Universal Robots PolyScope program: OnRobot_Pin_Insertion_Example.urp

Program OnRobot_Pin_Insertion_Example (createdIn=3.3.4.310 lastSavedIn=3.7.0.40195 robotSerialNumber=2014359999 directory=/home/ur/ursim-current/programs/TransferVM/Examples/Pendrive installation=default)
Calibrated DH parameters: a=[0.000125, -0.611383, -0.570393, -0.000092, 0.000088, 0]; d=[0.127903, 2.433032, -6.959421, 4.690192, 0.11563, 0.092223]; alpha=[1.570378, -0.01465, -0.007405, 1.570477, -1.570381, 0]; deltaTheta=[-0.000064, -0.058226, 0.116976, -0.058728, 0.000029, -0.000013]
BeforeStart
  URCap F/T Zero (FT-OnRobot, OnRobot A/S)
Robot Program (runOnlyOnce=true)
  URCap F/T Guard (FT-OnRobot, OnRobot A/S) dataModel(OF_PID=0, FX=0.0, FY=0.0, FZ=0.0, TX=0.0, TY=0.0, TZ=0.0, F3D=50.0, T3D=1.0, ABS=true, COORD=0, INDEX=0, STATE=true, ADVANCED=false, NEEDDIGI=false, NAME=50N & 1Nm)
    MoveJ speed 60 deg/s, acceleration 80 deg/s^2 (useActiveTCP=false)
      Waypoint StartWP: TCP in base x=-120.113 y=-431.763 z=146.073 mm, rx=-0.0012 ry=3.1163 rz=0.0389 rad; joints [-91.713, -98.956, -126.223, -46.295, 91.393, -1.776] deg
    URCap F/T Insert Part (FT-OnRobot, OnRobot A/S) dataModel(SPEED=0.05, DEPTH=0.02, FORCE=3, TORQUE=0.2, NAME=20 mm, LEN=0, DEG=0, SILENT=false, ADVANCED=false, ASTART=10, AEND=30, ALIMIT=0.17453292519943295, ASTRENGTH=0.5, pushingForce=5.0, minDistance=0.02, maxDistance=0.042, advanced=true, generateWarning=true, fx=0.0, cfx=true, fy=0.0, cfy=true, fz=0.0, cfz=true, tx=0.0, ctx=true, ty=0.0, cty=true, ctz=true, tz=0.0)
    If (of_return == 0)  or  (of_return == 1) or (of_return == 2)
      Popup Message (haltProgram=false message=Pin insertion was successful!)
    Else 
      Popup Message (haltProgram=false message=Pin insertion was not successful!)
    URCap F/T Control (FT-OnRobot, OnRobot A/S) dataModel(coordsys=1, name=Pin release, enarray=[true, true, false, false, false, false])
      URCap F/T Move (FT-OnRobot, OnRobot A/S) dataModel(coordsys=1, absolute=false, speed=0.025, acceleration=0.5, rpy=[0.0, 0.0, 0.0], popupLimit=false, ftarray=[0.0, 0.0, 0.0, 0.0, 0.0, 0.0, 50.0, 0.0], ftabsarray=[false, false, false, false, false, false])
        URCap F/T Waypoint (FT-OnRobot, OnRobot A/S) dataModel(relativeCoords=[0.0, 0.0, -0.055, 0.0, 0.0, 0.0], type=2, z=-0.05)
